PROGRAM SystemClock
VAR
	ton_RefreshTime			: TON :=(PT:= T#10mS);
	fb_GetLocalSystemtime 	: FB_localSystemTime;
	s_systemDateTime		: STRING(40);
END_VAR

ton_RefreshTime(IN:= NOT(ton_RefreshTime.Q));

IF ton_RefreshTime.Q THEN
	fb_GetLocalSystemtime(
		bEnable := TRUE,
		dwCycle := 1);
	s_SystemDateTime := SYSTEMTIME_TO_STRING(fb_GetLocalSystemtime.systemTime);
	gvl.dt_SystemDateTime := SYSTEMTIME_TO_DT(fb_GetLocalSystemtime.systemTime);
	GVL.s_SystemDate := MID(s_SystemDateTime, 10, 1);
	GVL.s_SystemTime := MID(s_SystemDateTime, 12, 12);
END_IF

GVL.b_SystemClockOK := GVL.s_SystemDate <> '1970-01-01' AND GVL.s_SystemTime <> '00:00:00';

END_PROGRAM

(* stored: Version 1.1.0.1, ProductVersion 3.1.4026.18
   POU SystemClock: Id {0caa7ee7-18d6-436d-ba58-a44e5b5f4705}, SpecialFunc None *)
